	E_State.ReadTable:
		// Mover 1 stays where it is. Ask the NC what slave position the table wants for it.
		// The table master runs from TABLE_START to TABLE_START + 1500, so a track position
		// below the table start is one lap further on in the table.
		IF NOT fbReadTable.Execute THEN
			fMasterInTable := fMover1Pos;
			IF fMasterInTable < TABLE_START THEN
				fMasterInTable := fMasterInTable + TRACK_LENGTH;
			END_IF
			fbReadTable.CamTableID := CAM_TABLE_ID;
			fbReadTable.MasterPosition := fMasterInTable;
		END_IF
		fbReadTable.Execute := TRUE;
		IF fbReadTable.Done THEN
			fbReadTable.Execute := FALSE;
			// table: slave = master - gap   ->   gap = master - slave
			fGapWanted := fMasterInTable - fbReadTable.SlavePosition;
			// Mover 1 stands still, so this relative move can never run into it:
			// positive = Mover 2 closes up from behind, negative = Mover 2 backs off a little
			fbMoveRelMover2.Distance := fGapActual - fGapWanted;
			eState := E_State.Preposition;
		END_IF

	E_State.Preposition:
		fbMoveRelMover2.Velocity := POSITIONING_VELOCITY;
		fbMoveRelMover2.Execute := TRUE;
		IF fbMoveRelMover2.Done THEN
			fbMoveRelMover2.Execute := FALSE;
			eState := E_State.CamIn;
		END_IF

	E_State.CamIn:
		fbCamIn.CamTableID := CAM_TABLE_ID;
		fbCamIn.StartMode := MC_STARTMODE_ABSOLUTE;		// table master axis = Mover 1 track position
		fbCamIn.MasterOffset := 0.0;
		fbCamIn.SlaveOffset := 0.0;
		fbCamIn.MasterScaling := 1.0;
		fbCamIn.SlaveScaling := 1.0;
		// let the NC pick the slave offset so Mover 2 never jumps at coupling.
		// After the pre-positioning above that offset is 0 (or whole laps), so the table gaps apply 1:1.
		fbCamIn.Options.SlaveScalingMode := MC_CAMSCALING_AUTOOFFSET;
		fbCamIn.Execute := TRUE;
		IF fbCamIn.InSync THEN
			fbCamIn.Execute := FALSE;
			eState := E_State.Run;
		END_IF

	E_State.Run:
		// only the master is commanded - the slave is driven by the cam
		fbMoveVeloMover1.Velocity := MASTER_VELOCITY;
		fbMoveVeloMover1.Direction := MC_Positive_Direction;
		fbMoveVeloMover1.Execute := TRUE;
		IF bStop THEN
			bStop := FALSE;
			fbMoveVeloMover1.Execute := FALSE;
			eState := E_State.Stopping;
		END_IF

	E_State.Stopping:
		fbHaltMover1.Execute := TRUE;
		IF fbHaltMover1.Done THEN
			fbHaltMover1.Execute := FALSE;
			eState := E_State.CamOut;
		END_IF

	E_State.CamOut:
		fbCamOut.Execute := TRUE;
		IF fbCamOut.Done THEN
			fbCamOut.Execute := FALSE;
			eState := E_State.Idle;
		END_IF

	E_State.Error:
		fbCamTableSelect.Execute := FALSE;
		fbReadTable.Execute := FALSE;
		fbMoveRelMover2.Execute := FALSE;
		fbCamIn.Execute := FALSE;
		fbMoveVeloMover1.Execute := FALSE;
		// a slave error does not stop the master: halt Mover 1 if it is still running and not in error itself
		fbHaltMover1.Execute := NOT GVL_Axes.Mover1.Status.Error AND GVL_Axes.Mover1.Status.Moving;
		fbCamOut.Execute := FALSE;
		IF bReset THEN
			bReset := FALSE;
			fbResetMover1.Execute := TRUE;
			fbResetMover2.Execute := TRUE;
			eState := E_State.Resetting;
		END_IF

	E_State.Resetting:
		IF (fbResetMover1.Done OR fbResetMover1.Error) AND (fbResetMover2.Done OR fbResetMover2.Error) THEN
			fbResetMover1.Execute := FALSE;
			fbResetMover2.Execute := FALSE;
			bError := FALSE;
			nErrorID := 0;
			sTableError := '';
			eState := E_State.Idle;
		END_IF
END_CASE

// any error anywhere -> Error state
IF eState <> E_State.Error AND eState <> E_State.Resetting THEN
	IF GVL_Axes.Mover1.Status.Error THEN
		nErrorID := GVL_Axes.Mover1.Status.ErrorID;
	ELSIF GVL_Axes.Mover2.Status.Error THEN
		nErrorID := GVL_Axes.Mover2.Status.ErrorID;
	ELSIF fbPowerMover1.Error THEN
		nErrorID := fbPowerMover1.ErrorID;
	ELSIF fbPowerMover2.Error THEN
		nErrorID := fbPowerMover2.ErrorID;
	ELSIF sTableError <> '' THEN
		nErrorID := PLC_ERROR_ID;
	ELSIF fbCamTableSelect.Error THEN
		nErrorID := fbCamTableSelect.ErrorID;
	ELSIF fbReadTable.Error THEN
		nErrorID := fbReadTable.ErrorID;
	ELSIF fbMoveRelMover2.Error THEN
		nErrorID := fbMoveRelMover2.ErrorID;
	ELSIF fbCamIn.Error THEN
		nErrorID := fbCamIn.ErrorID;
	ELSIF fbMoveVeloMover1.Error THEN
		nErrorID := fbMoveVeloMover1.ErrorID;
	ELSIF fbHaltMover1.Error THEN
		nErrorID := fbHaltMover1.ErrorID;
	ELSIF fbCamOut.Error THEN
		nErrorID := fbCamOut.ErrorID;
	END_IF
	IF nErrorID <> 0 THEN
		bError := TRUE;
		eState := E_State.Error;
	END_IF
END_IF

// call every function block once per cycle
fbPowerMover1(Axis := GVL_Axes.Mover1);
fbPowerMover2(Axis := GVL_Axes.Mover2);
fbResetMover1(Axis := GVL_Axes.Mover1);
fbResetMover2(Axis := GVL_Axes.Mover2);
fbCamTableSelect(Master := GVL_Axes.Mover1, Slave := GVL_Axes.Mover2, CamTable := stCamTable);
fbReadTable();
fbMoveRelMover2(Axis := GVL_Axes.Mover2);
fbCamIn(Master := GVL_Axes.Mover1, Slave := GVL_Axes.Mover2);
fbMoveVeloMover1(Axis := GVL_Axes.Mover1);
fbHaltMover1(Axis := GVL_Axes.Mover1);
fbCamOut(Slave := GVL_Axes.Mover2);

ACTION BuildCurveModule:
// ONE curve module as a module-relative cam piece: master 0..CURVE_TABLE_LENGTH measured from the module start,
// slave measured from the same origin with the ball gap included (point 1 = (0, -BALL_DISTANCE)). The same geometry
// as example 2, just for a single module at the origin: 8 clothoid points (ramp / plateau / ramp / line at the
// entry, mirrored at the exit) plus one 1:1 point at each end = 10 points.
//
// BuildTable pastes the 8 inner points wherever the layout says "Curve". Tuning the clothoid (the knot defaults
// in FB_XtsBallCamBuilder) happens here, once, independent of where the curves are on the track.
fbBuilder.fMasterStart		:= 0.0;
fbBuilder.fMasterEnd		:= CURVE_TABLE_LENGTH;
fbBuilder.fBallDistance		:= BALL_DISTANCE;
fbBuilder.fBallOffset		:= BALL_OFFSET;
fbBuilder.nCurves			:= 1;
fbBuilder.aCurveStart[1]	:= 0.0;
fbBuilder.fModuleLength		:= MODULE_LENGTH;
// fTransLength, aEntryKnots, aExitKnots keep the FB defaults (tuned for 115 mm / 103 mm on AT2050 modules)
fbBuilder.pPoints			:= ADR(aCurvePoints);
fbBuilder.nMaxPoints		:= MAX_CURVE_POINTS;

IF fbBuilder.Build() THEN
	nCurvePoints := fbBuilder.nPoints;		// 10
ELSE
	nCurvePoints := 0;
	sTableError := fbBuilder.sError;
END_IF
END_ACTION

ACTION BuildTable:
// The same table as example 2 (18 points, master TABLE_START .. +1500), assembled differently:
// the clothoid exists once, as a module-relative piece (BuildCurveModule -> aCurvePoints), and the track is a list
// of segments. FB_XtsCamStitcher walks the list, pastes the 8 inner curve points at every "Curve" (shifted by the
// running master position) and lets the straights run 1:1 without any points of their own.
// Changing a straight = changing a length in the list. The clothoid piece is untouched.
//
// Rules for the list: start and end on a straight (the table's first/last point must be 1:1), and every straight
// after a curve must be longer than the curve piece overhangs the module (103 mm with the default knots). The
// stitcher reports an error otherwise.
sTableError := '';
nCamPoints := 0;

BuildCurveModule();
IF nCurvePoints = 0 THEN RETURN; END_IF		// sTableError is set

// one lap starting at TABLE_START (180): rest of straight 1 | curve 1 | straight 2 | curve 2 | start of straight 1
fbStitcher.aLayout[1].eKind := E_SegmentKind.Straight;	fbStitcher.aLayout[1].fLength := CURVE_1_START - TABLE_START;			//  70
fbStitcher.aLayout[2].eKind := E_SegmentKind.Curve;		fbStitcher.aLayout[2].fLength := MODULE_LENGTH;							// 500
fbStitcher.aLayout[3].eKind := E_SegmentKind.Straight;	fbStitcher.aLayout[3].fLength := CURVE_2_START - STRAIGHT_2_START;		// 250
fbStitcher.aLayout[4].eKind := E_SegmentKind.Curve;		fbStitcher.aLayout[4].fLength := MODULE_LENGTH;							// 500
fbStitcher.aLayout[5].eKind := E_SegmentKind.Straight;	fbStitcher.aLayout[5].fLength := TABLE_START - STRAIGHT_1_START;		// 180
fbStitcher.nSegments	:= 5;
fbStitcher.fMasterStart	:= TABLE_START;
fbStitcher.fStraightGap	:= BALL_DISTANCE;
fbStitcher.pCurvePoints	:= ADR(aCurvePoints[2]);	// the 8 clothoid points, without the 1:1 end points of the piece
fbStitcher.nCurvePoints	:= nCurvePoints - 2;
fbStitcher.pPoints		:= ADR(aCamPoints);
fbStitcher.nMaxPoints	:= MAX_CAM_POINTS;

IF NOT fbStitcher.Build() THEN
	sTableError := fbStitcher.sError;
	RETURN;
END_IF
IF ABS(fbStitcher.fLength - TRACK_LENGTH) > 0.001 THEN
	sTableError := 'layout does not add up to one lap';
	RETURN;
END_IF
nCamPoints := fbStitcher.nPoints;		// 18

// describe the array to the NC
stCamTable.pArray		:= ADR(aCamPoints);
stCamTable.ArraySize	:= nCamPoints * SIZEOF(MC_MotionFunctionPoint);
stCamTable.TableType	:= MC_TABLETYPE_MOTIONFUNCTION;
stCamTable.NoOfRows		:= nCamPoints;
stCamTable.NoOfColumns	:= 1;

// self-check: build the example 2 table next to it and compare point by point
fbBuilder.fMasterStart		:= TABLE_START;
fbBuilder.fMasterEnd		:= TABLE_START + TRACK_LENGTH;
fbBuilder.nCurves			:= 2;
fbBuilder.aCurveStart[1]	:= CURVE_1_START;
fbBuilder.aCurveStart[2]	:= CURVE_2_START;
fbBuilder.pPoints			:= ADR(aCheckPoints);
fbBuilder.nMaxPoints		:= MAX_CAM_POINTS;
fStitchMaxDeviation := 0.0;
IF fbBuilder.Build() AND_THEN fbBuilder.nPoints = nCamPoints THEN
	FOR i := 1 TO UDINT_TO_UINT(nCamPoints) DO
		fStitchMaxDeviation := MAX(fStitchMaxDeviation, ABS(aCamPoints[i].MasterPos - aCheckPoints[i].MasterPos));
		fStitchMaxDeviation := MAX(fStitchMaxDeviation, ABS(aCamPoints[i].SlavePos  - aCheckPoints[i].SlavePos));
	END_FOR
ELSE
	fStitchMaxDeviation := -1.0;		// could not compare
END_IF
END_ACTION

END_PROGRAM

// ---- POUs/FB_XtsCamStitcher.TcPOU
FUNCTION_BLOCK FB_XtsCamStitcher
(* Stitches a cam table (MC_MotionFunctionPoint array) for one lap of an XTS track out of segments:
     Straight - the cam runs 1:1 (slave = master - fStraightGap). Contributes no point of its own.
     Curve    - one 180 deg module, pasted from a module-relative point list: master AND slave measured from the
                module start, gap already included (e.g. the 8 inner points of PRG_Example3.aCurvePoints).
   The layout must start and end on a straight, and every straight after a curve must be longer than the curve
   points reach past the module end (103 mm with the default clothoid knots). Otherwise the master positions stop
   increasing and Build() reports an error. All SlaveVelo/SlaveAcc/SlaveJerk = 0, as in FB_XtsBallCamBuilder. *)
VAR CONSTANT
	MAX_SEGMENTS	: UINT := 8;
END_VAR
VAR_INPUT
	aLayout			: ARRAY[1..MAX_SEGMENTS] OF ST_CamSegment;	// the track, segment by segment, starting at fMasterStart
	nSegments		: UINT;					// entries of aLayout in use
	fMasterStart	: LREAL;				// [mm] master position of the first table point (must lie on a straight)
	fStraightGap	: LREAL;				// [mm] the slave trails the master by this much on a straight
	pCurvePoints	: POINTER TO MC_MotionFunctionPoint;	// module-relative points of ONE curve module
	nCurvePoints	: UDINT;				// number of those points
	pPoints			: POINTER TO MC_MotionFunctionPoint;	// target buffer: ADR(camPoints[first element])
	nMaxPoints		: UDINT;				// number of elements in the target buffer
END_VAR
VAR_OUTPUT
	nPoints			: UDINT;				// points written (use as NoOfRows)
	fLength			: LREAL;				// [mm] sum of the segment lengths = master range of the table
	bError			: BOOL;
	sError			: STRING(255);
END_VAR

(* nothing cyclic: call Build() once *)

METHOD PRIVATE AddPoint
VAR_INPUT
	fMaster	: LREAL;
	fSlave	: LREAL;
	eFunc	: MC_MotionFunctionType;
END_VAR
IF bError THEN RETURN; END_IF
IF nPoints >= nMaxPoints THEN
	bError := TRUE; sError := 'point buffer too small'; RETURN;
END_IF
IF nPoints > 0 AND_THEN fMaster <= pPoints[nPoints - 1].MasterPos THEN
	bError := TRUE;
	sError := CONCAT('master positions not increasing at point ', UDINT_TO_STRING(nPoints + 1));
	sError := CONCAT(sError, ' (a straight shorter than the curve overhang?)');
	RETURN;
END_IF

pPoints[nPoints].PointIndex        := nPoints + 1;
pPoints[nPoints].MasterPos         := fMaster;
pPoints[nPoints].SlavePos          := fSlave;
pPoints[nPoints].FunctionType      := eFunc;
pPoints[nPoints].PointType         := SEL(nPoints = 0, MC_MotionPointType.MOTIONPOINTTYPE_MOTION, MC_MotionPointType.MOTIONPOINTTYPE_ACTIVATION);
pPoints[nPoints].RelIndexNextPoint := 1;
pPoints[nPoints].SlaveVelo         := 0.0;
pPoints[nPoints].SlaveAcc          := 0.0;
pPoints[nPoints].SlaveJerk         := 0.0;
nPoints := nPoints + 1;
END_METHOD

METHOD Build : BOOL
VAR
	i	: UINT;
	k	: UDINT;
	fM	: LREAL;	// master position where the current segment starts
END_VAR
bError := FALSE; sError := ''; nPoints := 0; fLength := 0.0;

IF pPoints = 0 OR nMaxPoints < 2 THEN
	bError := TRUE; sError := 'pPoints / nMaxPoints not set'; RETURN;
END_IF
IF nSegments < 1 OR nSegments > MAX_SEGMENTS THEN
	bError := TRUE; sError := 'nSegments must be 1..8'; RETURN;
END_IF
IF aLayout[1].eKind <> E_SegmentKind.Straight OR aLayout[nSegments].eKind <> E_SegmentKind.Straight THEN
	bError := TRUE; sError := 'layout must start and end on a straight'; RETURN;
END_IF

// first point: on a straight, 1:1 line towards whatever comes next
fM := fMasterStart;
AddPoint(fM, fM - fStraightGap, MC_MotionFunctionType.MOTIONFUNCTYPE_POLYNOM1);

FOR i := 1 TO nSegments DO
	IF aLayout[i].eKind = E_SegmentKind.Curve THEN
		IF pCurvePoints = 0 OR nCurvePoints = 0 THEN
			bError := TRUE; sError := 'pCurvePoints / nCurvePoints not set'; RETURN;
		END_IF
		// paste the module: shift master and slave by the module start, keep the curve types
		FOR k := 0 TO nCurvePoints - 1 DO
			AddPoint(fM + pCurvePoints[k].MasterPos, fM + pCurvePoints[k].SlavePos, pCurvePoints[k].FunctionType);
		END_FOR
	END_IF
	// a straight adds nothing: the line from the previous point simply continues 1:1
	fM := fM + aLayout[i].fLength;
END_FOR
fLength := fM - fMasterStart;

// last point: back on a straight
AddPoint(fM, fM - fStraightGap, MC_MotionFunctionType.MOTIONFUNCTYPE_POLYNOM1);

IF NOT bError THEN
	pPoints[nPoints - 1].RelIndexNextPoint := 0;	// terminate the table
END_IF
Build := NOT bError;
END_METHOD

END_FUNCTION_BLOCK

// ---- POUs/PRG_Example4.TcPOU
// Example 4 - TwoTableSwitching: TWO cam tables that the NC swaps at the curve boundaries while running.
//
//   Mover 1 = master, runs at constant velocity around the track.
//   Mover 2 = slave, follows Mover 1 through whichever table is active.
//
// Table 1 (CAM_TABLE_ID)   = a 2-point straight line, Mover 2 BALL_DISTANCE behind Mover 1, periodic over one lap.
// Table 2 (CURVE_TABLE_ID) = the 10-point clothoid piece from BuildCurveModule, master 0..CURVE_TABLE_LENGTH from
//                            the module start.
// Neither table knows where the curves are. That is in aSwitch: while running, SwitchTables re-issues MC_CamIn
// four times per lap so the NC swaps tables at 250 / 870 / 1000 / 120 mm. Change the straights = change the
// switch positions, neither table is rebuilt.
//
// How to run (online view, with MAIN.eExample = TwoTableSwitching):  bStart -> watch eState -> bStop.   On Error: bReset.
// Watch fGapActual (115 on the straights), nActiveTableID (1/2) and nSwitchCount (+4 per lap).
PROGRAM PRG_Example4
VAR CONSTANT
	// --- track geometry (mm) ---
	TRACK_LENGTH			: LREAL := 1500.0;	// = modulo factor of both mover axes
	STRAIGHT_1_START		: LREAL := 0.0;
	CURVE_1_START			: LREAL := 250.0;
	STRAIGHT_2_START		: LREAL := 750.0;
	CURVE_2_START			: LREAL := 1000.0;
	MODULE_LENGTH			: LREAL := 500.0;	// one 180 deg curve module (AT2050)

	// --- the ball clamped between the two movers (see example 2) ---
	BALL_DISTANCE			: LREAL := 115.0;	// mm between the two jaws, measured along the ball's path
	BALL_OFFSET				: LREAL := 103.03;	// mm the ball (and the jaws) sit outboard of the mover path

	// --- the clothoid as ONE module-relative piece ---
	CURVE_TABLE_LENGTH		: LREAL := 620.0;	// mm of master one curve piece covers, measured from the module start.
												// Must reach past the builder's last exit knot (603): the trailing ball
												// keeps the cam busy 103 mm after the module ends. The builder errors if not.
	MAX_CURVE_POINTS		: UDINT := 16;

	// --- demo dynamics ---
	MASTER_VELOCITY			: LREAL := 300.0;	// mm/s, Mover 1 while running
	POSITIONING_VELOCITY	: LREAL := 200.0;	// mm/s, Mover 2 while pre-positioning

	CAM_TABLE_ID			: MC_CAM_ID := 1;	// NC > Tables > Table 1 (Ex 1-4) > Mover 2: the straight table
	CURVE_TABLE_ID			: MC_CAM_ID := 2;	// NC > Tables > Table 2 (Ex 4 curve) > Mover 2: the clothoid piece
	CAM_POINTS				: UDINT := 2;		// the straight table
	SWITCH_MISS_TOLERANCE	: LREAL := 50.0;	// mm Mover 1 may pass a queued switch position before the PLC calls it missed
	PLC_ERROR_ID			: UDINT := 16#FFFF_FFFF;	// not an NC error: the PLC side refused (builder, layout check,
													// missed table switch), see sTableError
END_VAR
VAR
	// --- commands: set TRUE in the online view, they reset themselves ---
	bStart				: BOOL;
	bStop				: BOOL;
	bReset				: BOOL;
	eState				: E_State;

	// --- table 1: the straight line, loaded into NC table CAM_TABLE_ID ---
	aCamPoints			: ARRAY[1..CAM_POINTS] OF MC_MotionFunctionPoint;
	stCamTable			: MC_CAM_REF;
	bTablesOk			: BOOL;			// BuildTable succeeded (FALSE with sTableError set: the PLC side refused)

	// --- table 2: the clothoid piece, loaded into NC table CURVE_TABLE_ID ---
	fbBuilder			: FB_XtsBallCamBuilder;	// computes the clothoid points of one module
	aCurvePoints		: ARRAY[1..MAX_CURVE_POINTS] OF MC_MotionFunctionPoint;	// 10 points, master 0..CURVE_TABLE_LENGTH from the module start
	nCurvePoints		: UDINT;
	stCurveTable		: MC_CAM_REF;
	fbCurveTableSelect	: MC_CamTableSelect;	// PLC array -> NC cam table CURVE_TABLE_ID

	// --- the switching ---
	fbCamSwitch			: MC_CamIn;		// re-couples Mover 2 to the other table when Mover 1 reaches a position (online table change)
	aSwitch				: ARRAY[1..4] OF ST_CamSwitch;	// the four switches of one lap, in track order
	nSwitch				: UINT;			// index of the switch queued next (0 = not initialised yet)
	fSwitchAxisPos		: LREAL;		// non-modulo Mover 1 position handed to the NC for the queued switch
	nActiveTableID		: MC_CAM_ID;	// the table driving Mover 2 right now
	nSwitchCount		: UDINT;		// switches done since coupling

	// --- function blocks ---
	fbPowerMover1		: MC_Power;
	fbPowerMover2		: MC_Power;
	fbResetMover1		: MC_Reset;
	fbResetMover2		: MC_Reset;
	fbCamTableSelect	: MC_CamTableSelect;			// PLC array -> NC cam table CAM_TABLE_ID
	fbReadTable			: MC_ReadCamTableSlaveDynamics;	// "where does the table want the slave for this master position?"
	fbMoveRelMover2		: MC_MoveRelative;
	fbCamIn				: MC_CamIn;
	fbMoveVeloMover1	: MC_MoveVelocity;
	fbHaltMover1		: MC_Halt;
	fbCamOut			: MC_CamOut;

	// --- live values worth watching ---
	fMover1Pos			: LREAL;	// modulo set position of Mover 1 (0..1500)
	fMover2Pos			: LREAL;	// modulo set position of Mover 2 (0..1500)
	fGapActual			: LREAL;	// how far Mover 2 is behind Mover 1 right now (along the track)
	fGapWanted			: LREAL;	// what the straight table asked for at coupling time (= BALL_DISTANCE)
	bError				: BOOL;
	nErrorID			: UDINT;
	sTableError			: STRING(255);	// why the PLC side refused: builder, layout check or missed switch (nErrorID = PLC_ERROR_ID)

	// --- scratch ---
	i					: UINT;
	fDist				: LREAL;
	fBest				: LREAL;
END_VAR

// update axis status every cycle
GVL_Axes.Mover1();
GVL_Axes.Mover2();

// live gap: Mover 1 position minus Mover 2 position, wrapped to 0..1500
fMover1Pos := GVL_Axes.Mover1.NcToPlc.ModuloSetPos;
fMover2Pos := GVL_Axes.Mover2.NcToPlc.ModuloSetPos;
fGapActual := fMover1Pos - fMover2Pos;
IF fGapActual < 0.0 THEN
	fGapActual := fGapActual + TRACK_LENGTH;
END_IF

CASE eState OF
	E_State.Idle:
		IF bStart THEN
			bStart := FALSE;
			eState := E_State.Enable;
		END_IF

	E_State.Enable:
		fbPowerMover1.Enable := TRUE;
		fbPowerMover1.Enable_Positive := TRUE;
		fbPowerMover1.Enable_Negative := TRUE;
		fbPowerMover2.Enable := TRUE;
		fbPowerMover2.Enable_Positive := TRUE;
		fbPowerMover2.Enable_Negative := TRUE;
		IF fbPowerMover1.Status AND fbPowerMover2.Status THEN
			eState := E_State.Decouple;
		END_IF

	E_State.Decouple:
		// An earlier run may have left Mover 2 coupled: the NC keeps the coupling through an axis error and MC_Reset
		// does not clear it. MC_CamTableSelect refuses to overwrite a table that a coupled axis is using (0x4A26).
		IF NOT fbCamOut.Execute THEN
			IF GVL_Axes.Mover2.Status.Coupled THEN
				fbCamOut.Execute := TRUE;
			ELSE
				eState := E_State.BuildTable;
			END_IF
		ELSIF fbCamOut.Done THEN
			fbCamOut.Execute := FALSE;
			eState := E_State.BuildTable;
		END_IF

	E_State.BuildTable:
		// fill both point arrays once, then hand the straight table to the NC (overwrites cam table CAM_TABLE_ID)
		IF NOT fbCamTableSelect.Execute THEN
			BuildTable();
		END_IF
		IF bTablesOk THEN		// FALSE: the PLC side refused, the error check below picks up sTableError
			fbCamTableSelect.Periodic := TRUE;		// one table = one lap, repeat forever
			fbCamTableSelect.CamTableID := CAM_TABLE_ID;
			fbCamTableSelect.Execute := TRUE;
			IF fbCamTableSelect.Done THEN
				fbCamTableSelect.Execute := FALSE;
				eState := E_State.BuildCurveTable;
			END_IF
		END_IF

	E_State.BuildCurveTable:
		// the clothoid piece goes into the second NC table
		fbCurveTableSelect.Periodic := TRUE;		// a late switch then repeats the piece instead of stopping Mover 2 at the table end
		fbCurveTableSelect.CamTableID := CURVE_TABLE_ID;
		fbCurveTableSelect.Execute := TRUE;
		IF fbCurveTableSelect.Done THEN
			fbCurveTableSelect.Execute := FALSE;
			eState := E_State.ReadTable;
		END_IF

	E_State.ReadTable:
		// Mover 1 stays where it is. Ask the NC what slave position the straight table wants for it.
		// The table master runs 0..1500 = the track, so Mover 1's track position goes in as it is.
		fbReadTable.CamTableID := CAM_TABLE_ID;
		fbReadTable.MasterPosition := fMover1Pos;
		fbReadTable.Execute := TRUE;
		IF fbReadTable.Done THEN
			fbReadTable.Execute := FALSE;
			// table: slave = master - gap   ->   gap = master - slave
			fGapWanted := fMover1Pos - fbReadTable.SlavePosition;
			// Mover 1 stands still, so this relative move can never run into it:
			// positive = Mover 2 closes up from behind, negative = Mover 2 backs off a little
			fbMoveRelMover2.Distance := fGapActual - fGapWanted;
			eState := E_State.Preposition;
		END_IF

	E_State.Preposition:
		fbMoveRelMover2.Velocity := POSITIONING_VELOCITY;
		fbMoveRelMover2.Execute := TRUE;
		IF fbMoveRelMover2.Done THEN
			fbMoveRelMover2.Execute := FALSE;
			eState := E_State.CamIn;
		END_IF

	E_State.CamIn:
		// couple to the straight table first, wherever Mover 1 stands. If that is inside a curve window the ball
		// distance is only right from the first switch on - harmless, the movers are 115 mm apart on the track.
		fbCamIn.CamTableID := CAM_TABLE_ID;
		fbCamIn.StartMode := MC_STARTMODE_ABSOLUTE;		// table master axis = Mover 1 track position
		fbCamIn.MasterOffset := 0.0;
		fbCamIn.SlaveOffset := 0.0;
		fbCamIn.MasterScaling := 1.0;
		fbCamIn.SlaveScaling := 1.0;
		// let the NC pick the slave offset so Mover 2 never jumps at coupling.
		// After the pre-positioning above that offset is 0 (or whole laps), so the table gap applies 1:1.
		fbCamIn.Options.SlaveScalingMode := MC_CAMSCALING_AUTOOFFSET;
		fbCamIn.Execute := TRUE;
		IF fbCamIn.InSync THEN
			fbCamIn.Execute := FALSE;
			// SwitchTables initialises itself on its first call
			nActiveTableID := CAM_TABLE_ID;
			nSwitch := 0;
			nSwitchCount := 0;
			fbCamSwitch.Execute := FALSE;
			eState := E_State.Run;
		END_IF

	E_State.Run:
		// only the master is commanded - the slave is driven by the cam
		fbMoveVeloMover1.Velocity := MASTER_VELOCITY;
		fbMoveVeloMover1.Direction := MC_Positive_Direction;
		fbMoveVeloMover1.Execute := TRUE;
		SwitchTables();		// keeps one table switch queued in the NC at all times
		IF bStop THEN
			bStop := FALSE;
			fbMoveVeloMover1.Execute := FALSE;
			fbCamSwitch.Execute := FALSE;
			eState := E_State.Stopping;
		END_IF

	E_State.Stopping:
		fbHaltMover1.Execute := TRUE;
		IF fbHaltMover1.Done THEN
			fbHaltMover1.Execute := FALSE;
			eState := E_State.CamOut;
		END_IF

	E_State.CamOut:
		fbCamOut.Execute := TRUE;
		IF fbCamOut.Done THEN
			fbCamOut.Execute := FALSE;
			eState := E_State.Idle;
		END_IF

	E_State.Error:
		fbCamTableSelect.Execute := FALSE;
		fbCurveTableSelect.Execute := FALSE;
		fbReadTable.Execute := FALSE;
		fbMoveRelMover2.Execute := FALSE;
		fbCamIn.Execute := FALSE;
		fbCamSwitch.Execute := FALSE;
		fbMoveVeloMover1.Execute := FALSE;
		// a slave error does not stop the master: halt Mover 1 if it is still running and not in error itself
		fbHaltMover1.Execute := NOT GVL_Axes.Mover1.Status.Error AND GVL_Axes.Mover1.Status.Moving;
		fbCamOut.Execute := FALSE;
		IF bReset THEN
			bReset := FALSE;
			fbResetMover1.Execute := TRUE;
			fbResetMover2.Execute := TRUE;
			eState := E_State.Resetting;
		END_IF

	E_State.Resetting:
		IF (fbResetMover1.Done OR fbResetMover1.Error) AND (fbResetMover2.Done OR fbResetMover2.Error) THEN
			fbResetMover1.Execute := FALSE;
			fbResetMover2.Execute := FALSE;
			bError := FALSE;
			nErrorID := 0;
			sTableError := '';
			eState := E_State.Idle;
		END_IF
END_CASE

// any error anywhere -> Error state
IF eState <> E_State.Error AND eState <> E_State.Resetting THEN
	IF GVL_Axes.Mover1.Status.Error THEN
		nErrorID := GVL_Axes.Mover1.Status.ErrorID;
	ELSIF GVL_Axes.Mover2.Status.Error THEN
		nErrorID := GVL_Axes.Mover2.Status.ErrorID;
	ELSIF fbPowerMover1.Error THEN
		nErrorID := fbPowerMover1.ErrorID;
	ELSIF fbPowerMover2.Error THEN
		nErrorID := fbPowerMover2.ErrorID;
	ELSIF sTableError <> '' THEN
		nErrorID := PLC_ERROR_ID;
	ELSIF fbCamTableSelect.Error THEN
		nErrorID := fbCamTableSelect.ErrorID;
	ELSIF fbCurveTableSelect.Error THEN
		nErrorID := fbCurveTableSelect.ErrorID;
	ELSIF fbReadTable.Error THEN
		nErrorID := fbReadTable.ErrorID;
	ELSIF fbMoveRelMover2.Error THEN
		nErrorID := fbMoveRelMover2.ErrorID;
	ELSIF fbCamIn.Error THEN
		nErrorID := fbCamIn.ErrorID;
	ELSIF fbCamSwitch.Error THEN
		nErrorID := fbCamSwitch.ErrorID;
	ELSIF fbMoveVeloMover1.Error THEN
		nErrorID := fbMoveVeloMover1.ErrorID;
	ELSIF fbHaltMover1.Error THEN
		nErrorID := fbHaltMover1.ErrorID;
	ELSIF fbCamOut.Error THEN
		nErrorID := fbCamOut.ErrorID;
	END_IF
	IF nErrorID <> 0 THEN
		bError := TRUE;
		eState := E_State.Error;
	END_IF
END_IF

// call every function block once per cycle
fbPowerMover1(Axis := GVL_Axes.Mover1);
fbPowerMover2(Axis := GVL_Axes.Mover2);
fbResetMover1(Axis := GVL_Axes.Mover1);
fbResetMover2(Axis := GVL_Axes.Mover2);
fbCamTableSelect(Master := GVL_Axes.Mover1, Slave := GVL_Axes.Mover2, CamTable := stCamTable);
fbCurveTableSelect(Master := GVL_Axes.Mover1, Slave := GVL_Axes.Mover2, CamTable := stCurveTable);
fbReadTable();
fbMoveRelMover2(Axis := GVL_Axes.Mover2);
fbCamIn(Master := GVL_Axes.Mover1, Slave := GVL_Axes.Mover2);
fbCamSwitch(Master := GVL_Axes.Mover1, Slave := GVL_Axes.Mover2);
fbMoveVeloMover1(Axis := GVL_Axes.Mover1);
fbHaltMover1(Axis := GVL_Axes.Mover1);
fbCamOut(Slave := GVL_Axes.Mover2);

ACTION BuildCurveModule:
// ONE curve module as a module-relative cam piece: master 0..CURVE_TABLE_LENGTH measured from the module start,
// slave measured from the same origin with the ball gap included (point 1 = (0, -BALL_DISTANCE)). The same geometry
// as example 2, just for a single module at the origin: 8 clothoid points (ramp / plateau / ramp / line at the
// entry, mirrored at the exit) plus one 1:1 point at each end = 10 points.
//
// All 10 points go into NC table CURVE_TABLE_ID. Tuning the clothoid (the knot defaults in FB_XtsBallCamBuilder)
// happens here, once, independent of where the curves are on the track.
fbBuilder.fMasterStart		:= 0.0;
fbBuilder.fMasterEnd		:= CURVE_TABLE_LENGTH;
fbBuilder.fBallDistance		:= BALL_DISTANCE;
fbBuilder.fBallOffset		:= BALL_OFFSET;
fbBuilder.nCurves			:= 1;
fbBuilder.aCurveStart[1]	:= 0.0;
fbBuilder.fModuleLength		:= MODULE_LENGTH;
// fTransLength, aEntryKnots, aExitKnots keep the FB defaults (tuned for 115 mm / 103 mm on AT2050 modules)
fbBuilder.pPoints			:= ADR(aCurvePoints);
fbBuilder.nMaxPoints		:= MAX_CURVE_POINTS;

IF fbBuilder.Build() THEN
	nCurvePoints := fbBuilder.nPoints;		// 10
ELSE
	nCurvePoints := 0;
	sTableError := fbBuilder.sError;
END_IF
END_ACTION

ACTION BuildTable:
// Two NC tables instead of one:
//   table CAM_TABLE_ID   (1): a straight line, 2 points, Mover 2 BALL_DISTANCE behind Mover 1. Periodic over one lap.
//   table CURVE_TABLE_ID (2): the clothoid piece from BuildCurveModule, master 0..CURVE_TABLE_LENGTH from the module start.
// Neither table knows where the curves are. That is in aSwitch: while running, SwitchTables re-couples Mover 2 to
// the other table when Mover 1 reaches these positions.
//
// Only the straight table is "the" table for the start-up: ReadTable, Preposition and the first CamIn use it.
// The curve table is loaded in state BuildCurveTable.
sTableError := '';
bTablesOk := FALSE;

// table 1: the straight line
aCamPoints[1] := F_CamPoint(1, STRAIGHT_1_START, BALL_DISTANCE, MOTIONFUNCTYPE_POLYNOM1);	//    0: slave -115
aCamPoints[2] := F_CamPoint(2, TRACK_LENGTH,     BALL_DISTANCE, MOTIONFUNCTYPE_POLYNOM1);	// 1500: slave 1385, lift 1500 per lap
aCamPoints[2].RelIndexNextPoint := 0;
stCamTable.pArray		:= ADR(aCamPoints);
stCamTable.ArraySize	:= SIZEOF(aCamPoints);
stCamTable.TableType	:= MC_TABLETYPE_MOTIONFUNCTION;
stCamTable.NoOfRows		:= CAM_POINTS;
stCamTable.NoOfColumns	:= 1;

// table 2: the clothoid piece
BuildCurveModule();		// -> aCurvePoints / nCurvePoints (sTableError set if it refused)
IF nCurvePoints = 0 THEN RETURN; END_IF
stCurveTable.pArray			:= ADR(aCurvePoints);
stCurveTable.ArraySize		:= nCurvePoints * SIZEOF(MC_MotionFunctionPoint);
stCurveTable.TableType		:= MC_TABLETYPE_MOTIONFUNCTION;
stCurveTable.NoOfRows		:= nCurvePoints;
stCurveTable.NoOfColumns	:= 1;

// the four switches of a lap, in track order. The curve piece covers CURVE_TABLE_LENGTH from each module start, so
// the switch back to the straight table comes 120 mm into the following straight (curve 2: after the 1500 -> 0 wrap).
aSwitch[1].fTrackPos := CURVE_1_START;										aSwitch[1].nTableID := CURVE_TABLE_ID;	//  250
aSwitch[2].fTrackPos := CURVE_1_START + CURVE_TABLE_LENGTH;					aSwitch[2].nTableID := CAM_TABLE_ID;	//  870
aSwitch[3].fTrackPos := CURVE_2_START;										aSwitch[3].nTableID := CURVE_TABLE_ID;	// 1000
aSwitch[4].fTrackPos := CURVE_2_START + CURVE_TABLE_LENGTH - TRACK_LENGTH;	aSwitch[4].nTableID := CAM_TABLE_ID;	//  120

// the two curve pieces must not overlap: every straight has to be longer than the overhang (CURVE_TABLE_LENGTH - MODULE_LENGTH)
IF CURVE_TABLE_LENGTH - MODULE_LENGTH >= MIN(CURVE_2_START - STRAIGHT_2_START, CURVE_1_START + TRACK_LENGTH - (CURVE_2_START + MODULE_LENGTH)) THEN
	sTableError := 'curve pieces overlap - straights too short for two-table switching';
	RETURN;
END_IF

bTablesOk := TRUE;
END_ACTION

ACTION SwitchTables:
// Called every cycle in Run. Keeps exactly one table switch queued in the NC: MC_CamIn on an already coupled
// slave changes the table, and with Options.ActivationMode = ATMASTERAXISPOS the NC does it when Mover 1 passes
// Options.ActivationPosition. The PLC only has to be early, not exact. Both tables are 1:1 with gap BALL_DISTANCE
// at every switch position, so with SlaveScalingMode = AUTOOFFSET the position of Mover 2 does not jump and its
// velocity steps by ~1 % at most (the piece's 16 mm lead-in line has slope 1.0106, see README).
//
// Written against the Tc2_MC2_Camming 3.4.8 interface. Two details to confirm on the first run (see README):
//   - ActivationPosition is given as the non-modulo axis position (NcToPlc.SetPos + distance to go).
//   - MC_STARTMODE_RELATIVE: table master 0 = Mover 1 position at activation (= the module start for table 2).
IF nSwitch = 0 THEN
	// first call after coupling: start with the switch closest ahead of Mover 1
	// (a switch to the table that is already active is harmless)
	fBest := TRACK_LENGTH + 1.0;
	FOR i := 1 TO 4 DO
		fDist := aSwitch[i].fTrackPos - fMover1Pos;
		IF fDist <= 0.0 THEN fDist := fDist + TRACK_LENGTH; END_IF
		IF fDist < fBest THEN fBest := fDist; nSwitch := i; END_IF
	END_FOR
END_IF

IF NOT fbCamSwitch.Execute THEN
	// queue the next switch
	fDist := aSwitch[nSwitch].fTrackPos - fMover1Pos;
	IF fDist <= 0.0 THEN fDist := fDist + TRACK_LENGTH; END_IF
	fSwitchAxisPos := GVL_Axes.Mover1.NcToPlc.SetPos + fDist;
	fbCamSwitch.CamTableID := aSwitch[nSwitch].nTableID;
	fbCamSwitch.StartMode := MC_STARTMODE_RELATIVE;
	fbCamSwitch.MasterOffset := 0.0;
	fbCamSwitch.SlaveOffset := 0.0;
	fbCamSwitch.MasterScaling := 1.0;
	fbCamSwitch.SlaveScaling := 1.0;
	fbCamSwitch.Options.SlaveScalingMode := MC_CAMSCALING_AUTOOFFSET;
	fbCamSwitch.Options.ActivationMode := MC_CAMACTIVATION_ATMASTERAXISPOS;
	fbCamSwitch.Options.ActivationPosition := fSwitchAxisPos;
	fbCamSwitch.Execute := TRUE;
ELSIF fbCamSwitch.InSync THEN
	// the NC has switched
	fbCamSwitch.Execute := FALSE;
	nActiveTableID := aSwitch[nSwitch].nTableID;
	nSwitchCount := nSwitchCount + 1;
	nSwitch := nSwitch MOD 4 + 1;
ELSIF GVL_Axes.Mover1.NcToPlc.SetPos > fSwitchAxisPos + SWITCH_MISS_TOLERANCE THEN
	// Mover 1 is well past the position and the NC did not switch - stop rather than run the wrong table
	sTableError := 'cam table switch missed';		// -> PLC_ERROR_ID
END_IF
END_ACTION

END_PROGRAM

// ---- POUs/PRG_Example5.TcPOU
// Example 5 - VirtualMasterSplit: the BALL is the master. A virtual axis runs along the ball's path at constant
// velocity and BOTH movers follow it, each through its own cam table (10 points each from FB_XtsBallCamBuilder).
//
//   VirtualMaster = the ball. Its position is the distance the ball has travelled along its own path. That path
//                   lies BALL_OFFSET outboard of the track, so one lap of the ball is TRACK_LENGTH + 2*pi*BALL_OFFSET
//                   = 2147.36 mm (fBallLap), not 1500.
//   Mover 1       = slave of the virtual master. Its jaw sits BALL_DISTANCE/2 ahead of the ball along that path.
//   Mover 2       = slave of the virtual master. Its jaw sits BALL_DISTANCE/2 behind the ball.
//
// In example 2 Mover 1 ran at constant speed and Mover 2 did all the work: 178 % of Mover 1's speed going into a
// curve, 56 % coming out. Here the ball runs at constant speed instead. On the straights both movers run at the
// ball's speed. While a mover's jaw is in a curve the ball travels further than the mover (its path is longer), so
// that mover runs at 56 % of the ball's speed. Each mover slows down exactly while ITS jaw is in the curvature ramp
// of the module, so the two tables are the same curve shifted by BALL_DISTANCE along the master, and neither mover
// ever has to run faster than the ball.
//
// How to run (online view, with MAIN.eExample = VirtualMasterSplit):  bStart -> watch eState -> bStop.   On Error: bReset.
// Watch fGapActual (115 on the straights, dipping through the curves as in example 2) and fRatioMover1 / fRatioMover2
// (1.0 on the straights, 0.56 while that mover's jaw is in a curve, Mover 1 first, Mover 2 a moment later).
PROGRAM PRG_Example5
VAR CONSTANT
	// --- track geometry (mm) ---
	TRACK_LENGTH			: LREAL := 1500.0;	// = modulo factor of both mover axes
	CURVE_1_START			: LREAL := 250.0;
	CURVE_2_START			: LREAL := 1000.0;
	MODULE_LENGTH			: LREAL := 500.0;	// one 180 deg curve module (AT2050)

	// --- the ball clamped between the two movers (see example 2) ---
	BALL_DISTANCE			: LREAL := 115.0;	// mm between the two jaws, measured along the ball's path
	BALL_OFFSET				: LREAL := 103.03;	// mm the ball (and the jaws) sit outboard of the mover path
	TABLE_START				: LREAL := 125.0;	// track position of the ball at the first table point. Any point on
												// straight 1 that keeps both tables clear of the 1500 -> 0 wrap works
												// (57.5 < x < 192.5: Mover 1's jaw must still be before curve 1, Mover 2's
												// last exit ramp must end before the table does).

	// --- demo dynamics ---
	MASTER_VELOCITY			: LREAL := 300.0;	// mm/s, the ball while running (= the movers' speed on the straights)
	POSITIONING_VELOCITY	: LREAL := 200.0;	// mm/s, Mover 2 while pre-positioning

	MOVER1_TABLE_ID			: MC_CAM_ID := 3;	// NC > Tables > Table 3 (Ex 5 Mover 1) > Mover 1  (VirtualMaster -> Mover 1)
	MOVER2_TABLE_ID			: MC_CAM_ID := 4;	// NC > Tables > Table 4 (Ex 5 Mover 2) > Mover 2  (VirtualMaster -> Mover 2)
	MAX_CAM_POINTS			: UDINT := 16;		// the builder writes 4 per curve + 2 = 10 per table
	PLC_ERROR_ID			: UDINT := 16#FFFF_FFFF;	// not an NC error: the builder refused, see sTableError
END_VAR
VAR
	// --- commands: set TRUE in the online view, they reset themselves ---
	bStart				: BOOL;
	bStop				: BOOL;
	bReset				: BOOL;
	eState				: E_State;

	// --- cam table data: one table per mover, both with the ball as master ---
	aMover1Points		: ARRAY[1..MAX_CAM_POINTS] OF MC_MotionFunctionPoint;	// -> NC table MOVER1_TABLE_ID
	aMover2Points		: ARRAY[1..MAX_CAM_POINTS] OF MC_MotionFunctionPoint;	// -> NC table MOVER2_TABLE_ID
	nMover1Points		: UDINT;		// points actually used (10)
	nMover2Points		: UDINT;		// points actually used (10)
	stMover1Table		: MC_CAM_REF;
	stMover2Table		: MC_CAM_REF;
	bTablesOk			: BOOL;			// BuildTable succeeded (FALSE with sTableError set: the builder refused)
	fbBuilder			: FB_XtsBallCamBuilder;	// computes the points; also used to convert Mover 1's position into a ball position
	fBallLap			: LREAL;		// mm the ball travels per lap of the track = master period of both tables (2147.36)
	fTableMasterStart	: LREAL;		// ball position of the first table point (= TABLE_START, the ball is still on the straight)

	// --- function blocks ---
	fbPowerMover1		: MC_Power;
	fbPowerMover2		: MC_Power;
	fbPowerMaster		: MC_Power;
	fbResetMover1		: MC_Reset;
	fbResetMover2		: MC_Reset;
	fbResetMaster		: MC_Reset;
	fbTableSelectMover1	: MC_CamTableSelect;			// PLC array -> NC cam table MOVER1_TABLE_ID
	fbTableSelectMover2	: MC_CamTableSelect;			// PLC array -> NC cam table MOVER2_TABLE_ID
	fbSetMasterPos		: MC_SetPosition;				// puts the virtual master where the ball is for Mover 1's position
	fbReadTableMover1	: MC_ReadCamTableSlaveDynamics;	// "where does table 3 want Mover 1 for this ball position?"
	fbReadTableMover2	: MC_ReadCamTableSlaveDynamics;	// "where does table 4 want Mover 2 for this ball position?"
	fbMoveRelMover2		: MC_MoveRelative;
	fbCamInMover1		: MC_CamIn;
	fbCamInMover2		: MC_CamIn;
	fbMoveVeloMaster	: MC_MoveVelocity;
	fbHaltMaster		: MC_Halt;
	fbCamOutMover1		: MC_CamOut;
	fbCamOutMover2		: MC_CamOut;

	// --- live values worth watching ---
	fMover1Pos			: LREAL;	// modulo set position of Mover 1 (0..1500)
	fMover2Pos			: LREAL;	// modulo set position of Mover 2 (0..1500)
	fGapActual			: LREAL;	// how far Mover 2 is behind Mover 1 right now (along the track)
	fGapWanted			: LREAL;	// what the two tables asked for at coupling time
	fBallPos			: LREAL;	// where the ball is on its path in this lap (0..fBallLap, 0 = above track position 0)
	fMasterInTable		: LREAL;	// ball position handed to the NC at start-up, in the table's master range
	fAlignError			: LREAL;	// where table 3 wanted Mover 1 minus where it is, after AlignMaster (expect 0)
	fRatioMover1		: LREAL;	// Mover 1 speed / ball speed right now (1 on the straights, 0.56 in the arcs)
	fRatioMover2		: LREAL;	// Mover 2 speed / ball speed right now
	bError				: BOOL;
	nErrorID			: UDINT;
	sTableError			: STRING(255);	// why the builder refused (nErrorID = PLC_ERROR_ID)
END_VAR

// update axis status every cycle
GVL_Axes.Mover1();
GVL_Axes.Mover2();
GVL_Axes.VirtualMaster();

// live gap: Mover 1 position minus Mover 2 position, wrapped to 0..1500
fMover1Pos := GVL_Axes.Mover1.NcToPlc.ModuloSetPos;
fMover2Pos := GVL_Axes.Mover2.NcToPlc.ModuloSetPos;
fGapActual := fMover1Pos - fMover2Pos;
IF fGapActual < 0.0 THEN
	fGapActual := fGapActual + TRACK_LENGTH;
END_IF

// the virtual master is a linear axis (no modulo): wrap its position to one lap of the ball for display
IF fBallLap > 0.0 THEN
	fBallPos := GVL_Axes.VirtualMaster.NcToPlc.SetPos;
	fBallPos := fBallPos - fBallLap * DINT_TO_LREAL(TRUNC(fBallPos / fBallLap));
	IF fBallPos < 0.0 THEN
		fBallPos := fBallPos + fBallLap;
	END_IF
END_IF

// speed of each mover relative to the ball
IF ABS(GVL_Axes.VirtualMaster.NcToPlc.SetVelo) > 1.0 THEN
	fRatioMover1 := GVL_Axes.Mover1.NcToPlc.SetVelo / GVL_Axes.VirtualMaster.NcToPlc.SetVelo;
	fRatioMover2 := GVL_Axes.Mover2.NcToPlc.SetVelo / GVL_Axes.VirtualMaster.NcToPlc.SetVelo;
ELSE
	fRatioMover1 := 0.0;
	fRatioMover2 := 0.0;
END_IF

CASE eState OF
	E_State.Idle:
		IF bStart THEN
			bStart := FALSE;
			eState := E_State.Enable;
		END_IF

	E_State.Enable:
		fbPowerMover1.Enable := TRUE;
		fbPowerMover1.Enable_Positive := TRUE;
		fbPowerMover1.Enable_Negative := TRUE;
		fbPowerMover2.Enable := TRUE;
		fbPowerMover2.Enable_Positive := TRUE;
		fbPowerMover2.Enable_Negative := TRUE;
		fbPowerMaster.Enable := TRUE;
		fbPowerMaster.Enable_Positive := TRUE;
		fbPowerMaster.Enable_Negative := TRUE;
		IF fbPowerMover1.Status AND fbPowerMover2.Status AND fbPowerMaster.Status THEN
			eState := E_State.Decouple;
		END_IF

	E_State.Decouple:
		// An earlier run may have left a mover coupled: the NC keeps the coupling through an axis error and MC_Reset
		// does not clear it. MC_CamTableSelect refuses to overwrite a table that a coupled axis is using (0x4A26).
		IF NOT fbCamOutMover1.Execute AND NOT fbCamOutMover2.Execute THEN
			IF GVL_Axes.Mover1.Status.Coupled OR GVL_Axes.Mover2.Status.Coupled THEN
				fbCamOutMover1.Execute := GVL_Axes.Mover1.Status.Coupled;
				fbCamOutMover2.Execute := GVL_Axes.Mover2.Status.Coupled;
			ELSE
				eState := E_State.BuildTable;
			END_IF
		ELSIF (NOT fbCamOutMover1.Execute OR fbCamOutMover1.Done) AND (NOT fbCamOutMover2.Execute OR fbCamOutMover2.Done) THEN
			fbCamOutMover1.Execute := FALSE;
			fbCamOutMover2.Execute := FALSE;
			eState := E_State.BuildTable;
		END_IF

	E_State.BuildTable:
		// fill both point arrays once, then hand Mover 1's table to the NC (overwrites cam table MOVER1_TABLE_ID)
		IF NOT fbTableSelectMover1.Execute THEN
			BuildTable();
		END_IF
		IF bTablesOk THEN		// FALSE: the builder refused, the error check below picks up sTableError
			fbTableSelectMover1.Periodic := TRUE;		// one table = one lap of the ball, repeat forever
			fbTableSelectMover1.CamTableID := MOVER1_TABLE_ID;
			fbTableSelectMover1.Execute := TRUE;
			IF fbTableSelectMover1.Done THEN
				fbTableSelectMover1.Execute := FALSE;
				eState := E_State.LoadMover2Table;
			END_IF
		END_IF

	E_State.LoadMover2Table:
		// Mover 2's table goes into the second NC table
		fbTableSelectMover2.Periodic := TRUE;
		fbTableSelectMover2.CamTableID := MOVER2_TABLE_ID;
		fbTableSelectMover2.Execute := TRUE;
		IF fbTableSelectMover2.Done THEN
			fbTableSelectMover2.Execute := FALSE;
			eState := E_State.AlignMaster;
		END_IF

	E_State.AlignMaster:
		// Mover 1 stays where it is. The virtual master has no idea where the ball is, so tell it: Mover 1's jaw is at
		// track position fMover1Pos, which is BallArc(fMover1Pos) along the ball's path, and the ball itself is half a
		// ball distance behind the jaw. A value below the table start is one lap further on in the table.
		IF NOT fbSetMasterPos.Execute THEN
			fMasterInTable := fbBuilder.BallArc(fMover1Pos) - BALL_DISTANCE / 2.0;
			IF fMasterInTable < fTableMasterStart THEN
				fMasterInTable := fMasterInTable + fBallLap;
			END_IF
			fbSetMasterPos.Position := fMasterInTable;
			fbSetMasterPos.Mode := FALSE;		// absolute
		END_IF
		fbSetMasterPos.Execute := TRUE;
		IF fbSetMasterPos.Done THEN
			fbSetMasterPos.Execute := FALSE;
			eState := E_State.ReadTable;
		END_IF

	E_State.ReadTable:
		// Ask the NC where both tables want their mover for this ball position, one table after the other.
		// Table 3 should want Mover 1 exactly where it is (fAlignError = 0). Table 4 says where Mover 2 has to go.
		fbReadTableMover1.CamTableID := MOVER1_TABLE_ID;
		fbReadTableMover1.MasterPosition := fMasterInTable;
		fbReadTableMover1.Execute := TRUE;
		IF fbReadTableMover1.Done THEN
			fbReadTableMover2.CamTableID := MOVER2_TABLE_ID;
			fbReadTableMover2.MasterPosition := fMasterInTable;
			fbReadTableMover2.Execute := TRUE;
			IF fbReadTableMover2.Done THEN
				fbReadTableMover1.Execute := FALSE;
				fbReadTableMover2.Execute := FALSE;
				// both slave positions are track positions in the same lap, so their difference is the gap
				fGapWanted := fbReadTableMover1.SlavePosition - fbReadTableMover2.SlavePosition;
				// self-check: table 3 minus Mover 1, wrapped to -750..750 (whole laps do not count)
				fAlignError := fbReadTableMover1.SlavePosition - fMover1Pos;
				fAlignError := fAlignError - TRACK_LENGTH * DINT_TO_LREAL(TRUNC(fAlignError / TRACK_LENGTH));
				IF fAlignError > 0.5 * TRACK_LENGTH THEN fAlignError := fAlignError - TRACK_LENGTH; END_IF
				IF fAlignError < -0.5 * TRACK_LENGTH THEN fAlignError := fAlignError + TRACK_LENGTH; END_IF
				// Mover 1 stands still, so this relative move can never run into it:
				// positive = Mover 2 closes up from behind, negative = Mover 2 backs off a little
				fbMoveRelMover2.Distance := fGapActual - fGapWanted;
				eState := E_State.Preposition;
			END_IF
		END_IF

	E_State.Preposition:
		fbMoveRelMover2.Velocity := POSITIONING_VELOCITY;
		fbMoveRelMover2.Execute := TRUE;
		IF fbMoveRelMover2.Done THEN
			fbMoveRelMover2.Execute := FALSE;
			eState := E_State.CamIn;
		END_IF

	E_State.CamIn:
		// couple both movers to the virtual master, each through its own table
		fbCamInMover1.CamTableID := MOVER1_TABLE_ID;
		fbCamInMover1.StartMode := MC_STARTMODE_ABSOLUTE;		// table master axis = the virtual master's position
		fbCamInMover1.MasterOffset := 0.0;
		fbCamInMover1.SlaveOffset := 0.0;
		fbCamInMover1.MasterScaling := 1.0;
		fbCamInMover1.SlaveScaling := 1.0;
		// let the NC pick the slave offsets so that nobody jumps at coupling. After AlignMaster and the pre-positioning
		// both offsets are 0 (or whole laps), so the two tables apply 1:1 and the curves are where the track has them.
		fbCamInMover1.Options.SlaveScalingMode := MC_CAMSCALING_AUTOOFFSET;
		fbCamInMover2.CamTableID := MOVER2_TABLE_ID;
		fbCamInMover2.StartMode := MC_STARTMODE_ABSOLUTE;
		fbCamInMover2.MasterOffset := 0.0;
		fbCamInMover2.SlaveOffset := 0.0;
		fbCamInMover2.MasterScaling := 1.0;
		fbCamInMover2.SlaveScaling := 1.0;
		fbCamInMover2.Options.SlaveScalingMode := MC_CAMSCALING_AUTOOFFSET;
		fbCamInMover1.Execute := TRUE;
		fbCamInMover2.Execute := TRUE;
		IF fbCamInMover1.InSync AND fbCamInMover2.InSync THEN
			fbCamInMover1.Execute := FALSE;
			fbCamInMover2.Execute := FALSE;
			eState := E_State.Run;
		END_IF

	E_State.Run:
		// only the ball is commanded - both movers are driven by their cams
		fbMoveVeloMaster.Velocity := MASTER_VELOCITY;
		fbMoveVeloMaster.Direction := MC_Positive_Direction;
		fbMoveVeloMaster.Execute := TRUE;
		IF bStop THEN
			bStop := FALSE;
			fbMoveVeloMaster.Execute := FALSE;
			eState := E_State.Stopping;
		END_IF

	E_State.Stopping:
		fbHaltMaster.Execute := TRUE;
		IF fbHaltMaster.Done THEN
			fbHaltMaster.Execute := FALSE;
			eState := E_State.CamOut;
		END_IF

	E_State.CamOut:
		fbCamOutMover1.Execute := TRUE;
		fbCamOutMover2.Execute := TRUE;
		IF fbCamOutMover1.Done AND fbCamOutMover2.Done THEN
			fbCamOutMover1.Execute := FALSE;
			fbCamOutMover2.Execute := FALSE;
			eState := E_State.Idle;
		END_IF

	E_State.Error:
		fbTableSelectMover1.Execute := FALSE;
		fbTableSelectMover2.Execute := FALSE;
		fbSetMasterPos.Execute := FALSE;
		fbReadTableMover1.Execute := FALSE;
		fbReadTableMover2.Execute := FALSE;
		fbMoveRelMover2.Execute := FALSE;
		fbCamInMover1.Execute := FALSE;
		fbCamInMover2.Execute := FALSE;
		fbMoveVeloMaster.Execute := FALSE;
		// a slave error does not stop the master: halt the virtual master if it is still running and not in error itself
		fbHaltMaster.Execute := NOT GVL_Axes.VirtualMaster.Status.Error AND GVL_Axes.VirtualMaster.Status.Moving;
		fbCamOutMover1.Execute := FALSE;
		fbCamOutMover2.Execute := FALSE;
		IF bReset THEN
			bReset := FALSE;
			fbResetMover1.Execute := TRUE;
			fbResetMover2.Execute := TRUE;
			fbResetMaster.Execute := TRUE;
			eState := E_State.Resetting;
		END_IF

	E_State.Resetting:
		IF (fbResetMover1.Done OR fbResetMover1.Error) AND (fbResetMover2.Done OR fbResetMover2.Error)
			AND (fbResetMaster.Done OR fbResetMaster.Error) THEN
			fbResetMover1.Execute := FALSE;
			fbResetMover2.Execute := FALSE;
			fbResetMaster.Execute := FALSE;
			bError := FALSE;
			nErrorID := 0;
			sTableError := '';
			eState := E_State.Idle;
		END_IF
END_CASE

// any error anywhere -> Error state
IF eState <> E_State.Error AND eState <> E_State.Resetting THEN
	IF GVL_Axes.Mover1.Status.Error THEN
		nErrorID := GVL_Axes.Mover1.Status.ErrorID;
	ELSIF GVL_Axes.Mover2.Status.Error THEN
		nErrorID := GVL_Axes.Mover2.Status.ErrorID;
	ELSIF GVL_Axes.VirtualMaster.Status.Error THEN
		nErrorID := GVL_Axes.VirtualMaster.Status.ErrorID;
	ELSIF fbPowerMover1.Error THEN
		nErrorID := fbPowerMover1.ErrorID;
	ELSIF fbPowerMover2.Error THEN
		nErrorID := fbPowerMover2.ErrorID;
	ELSIF fbPowerMaster.Error THEN
		nErrorID := fbPowerMaster.ErrorID;
	ELSIF sTableError <> '' THEN
		nErrorID := PLC_ERROR_ID;
	ELSIF fbTableSelectMover1.Error THEN
		nErrorID := fbTableSelectMover1.ErrorID;
	ELSIF fbTableSelectMover2.Error THEN
		nErrorID := fbTableSelectMover2.ErrorID;
	ELSIF fbSetMasterPos.Error THEN
		nErrorID := fbSetMasterPos.ErrorID;
	ELSIF fbReadTableMover1.Error THEN
		nErrorID := fbReadTableMover1.ErrorID;
	ELSIF fbReadTableMover2.Error THEN
		nErrorID := fbReadTableMover2.ErrorID;
	ELSIF fbMoveRelMover2.Error THEN
		nErrorID := fbMoveRelMover2.ErrorID;
	ELSIF fbCamInMover1.Error THEN
		nErrorID := fbCamInMover1.ErrorID;
	ELSIF fbCamInMover2.Error THEN
		nErrorID := fbCamInMover2.ErrorID;
	ELSIF fbMoveVeloMaster.Error THEN
		nErrorID := fbMoveVeloMaster.ErrorID;
	ELSIF fbHaltMaster.Error THEN
		nErrorID := fbHaltMaster.ErrorID;
	ELSIF fbCamOutMover1.Error THEN
		nErrorID := fbCamOutMover1.ErrorID;
	ELSIF fbCamOutMover2.Error THEN
		nErrorID := fbCamOutMover2.ErrorID;
	END_IF
	IF nErrorID <> 0 THEN
		bError := TRUE;
		eState := E_State.Error;
	END_IF
END_IF

// call every function block once per cycle
fbPowerMover1(Axis := GVL_Axes.Mover1);
fbPowerMover2(Axis := GVL_Axes.Mover2);
fbPowerMaster(Axis := GVL_Axes.VirtualMaster);
fbResetMover1(Axis := GVL_Axes.Mover1);
fbResetMover2(Axis := GVL_Axes.Mover2);
fbResetMaster(Axis := GVL_Axes.VirtualMaster);
fbTableSelectMover1(Master := GVL_Axes.VirtualMaster, Slave := GVL_Axes.Mover1, CamTable := stMover1Table);
fbTableSelectMover2(Master := GVL_Axes.VirtualMaster, Slave := GVL_Axes.Mover2, CamTable := stMover2Table);
fbSetMasterPos(Axis := GVL_Axes.VirtualMaster);
fbReadTableMover1();
fbReadTableMover2();
fbMoveRelMover2(Axis := GVL_Axes.Mover2);
fbCamInMover1(Master := GVL_Axes.VirtualMaster, Slave := GVL_Axes.Mover1);
fbCamInMover2(Master := GVL_Axes.VirtualMaster, Slave := GVL_Axes.Mover2);
fbMoveVeloMaster(Axis := GVL_Axes.VirtualMaster);
fbHaltMaster(Axis := GVL_Axes.VirtualMaster);
fbCamOutMover1(Slave := GVL_Axes.Mover1);
fbCamOutMover2(Slave := GVL_Axes.Mover2);

ACTION BuildTable:
// Two tables with the same master: the ball. Master = distance the ball has travelled along its own path.
//   table MOVER1_TABLE_ID (3): where Mover 1 has to be so that its jaw is BALL_DISTANCE/2 AHEAD of the ball on that path.
//   table MOVER2_TABLE_ID (4): where Mover 2 has to be so that its jaw is BALL_DISTANCE/2 BEHIND the ball.
// The jaws are then BALL_DISTANCE apart along the ball's path, exactly as in example 2. Only the master changed:
// there it was Mover 1 (constant speed, Mover 2 did all the adjusting), here it is the ball.
//
// FB_XtsBallCamBuilder.BuildBallMaster does the geometry per mover: on a straight the mover runs at the ball's
// speed; while its jaw is in a curve module the ball's path (BALL_OFFSET outboard) is longer than the mover's, so
// the mover runs at 1/1.78 = 56 % of the ball's speed. The change happens exactly while the jaw is in the module's
// curvature ramp (84 mm of track), which is where the builder puts its knots: 4 points per curve (POLYNOM5 ramp,
// line on the arc, POLYNOM5 ramp, line on the straight) plus one point at each end = 10 points. No tuned knots.
//
// Both tables cover one lap of the track, from ball position TABLE_START (the ball is still on straight 1 there,
// so its path position equals the track position) to TABLE_START + fBallLap. Slave lift per lap: 1500, so the
// movers keep going around ("cyclic cam with lift").
sTableError := '';
bTablesOk := FALSE;
nMover1Points := 0;
nMover2Points := 0;

fbBuilder.fMasterStart		:= TABLE_START;
fbBuilder.fMasterEnd		:= TABLE_START + TRACK_LENGTH;
fbBuilder.fBallDistance		:= BALL_DISTANCE;
fbBuilder.fBallOffset		:= BALL_OFFSET;
fbBuilder.nCurves			:= 2;
fbBuilder.aCurveStart[1]	:= CURVE_1_START;
fbBuilder.aCurveStart[2]	:= CURVE_2_START;
fbBuilder.fModuleLength		:= MODULE_LENGTH;
// fTransLength keeps the FB default (84 mm, the AT2050 curvature ramp). The tuned knots are not used here.
fbBuilder.nMaxPoints		:= MAX_CAM_POINTS;

// table 3: Mover 1, jaw half a ball distance ahead of the ball
fbBuilder.pPoints := ADR(aMover1Points);
IF NOT fbBuilder.BuildBallMaster(fJawLead := BALL_DISTANCE / 2.0) THEN
	sTableError := fbBuilder.sError;
	RETURN;
END_IF
nMover1Points := fbBuilder.nPoints;		// 10

// table 4: Mover 2, jaw half a ball distance behind the ball
fbBuilder.pPoints := ADR(aMover2Points);
IF NOT fbBuilder.BuildBallMaster(fJawLead := -BALL_DISTANCE / 2.0) THEN
	sTableError := fbBuilder.sError;
	RETURN;
END_IF
nMover2Points := fbBuilder.nPoints;		// 10

// master range of the tables: one lap of the ball = 1500 + 2 pi * 103.03 = 2147.36 mm
fTableMasterStart	:= fbBuilder.BallArc(TABLE_START);
fBallLap			:= fbBuilder.BallArc(TABLE_START + TRACK_LENGTH) - fTableMasterStart;

// describe both arrays to the NC
stMover1Table.pArray		:= ADR(aMover1Points);
stMover1Table.ArraySize		:= nMover1Points * SIZEOF(MC_MotionFunctionPoint);
stMover1Table.TableType		:= MC_TABLETYPE_MOTIONFUNCTION;
stMover1Table.NoOfRows		:= nMover1Points;
stMover1Table.NoOfColumns	:= 1;

stMover2Table.pArray		:= ADR(aMover2Points);
stMover2Table.ArraySize		:= nMover2Points * SIZEOF(MC_MotionFunctionPoint);
stMover2Table.TableType		:= MC_TABLETYPE_MOTIONFUNCTION;
stMover2Table.NoOfRows		:= nMover2Points;
stMover2Table.NoOfColumns	:= 1;

bTablesOk := TRUE;
END_ACTION

END_PROGRAM
